PROGRAM Axis05_Auto
VAR
	Always_ON	:	BOOL	:=TRUE	;//상시 ON 
	Always_OFF	:	BOOL	:=FALSE	;//상시 OFF
END_VAR

// NETWORK 1

END_PROGRAM

(* stored: Version 1.1.0.1, ProductVersion 3.1.4024.15
   POU Axis05_Auto: Id {a556c58e-1b45-4a45-ad62-b9b9b34a80ae}, SpecialFunc None *)
